{attribute 'qualified_only'}
{attribute 'strict'}
TYPE E_MergeMode :
(
	BlockedWait := 0,
	Follow := 1,
	Lead := 2
);
END_TYPE

(* stored: Version 1.1.0.1, ProductVersion 3.1.4026.8
   DUT E_MergeMode: Id {57d55088-9666-061f-0842-13c5b7a7141d} *)
